FUNCTION_BLOCK PrintBools (* Basic Function Block Type *)
  (* Standard: 61499-2 *)
  (* Version 0.2, 2003-12-04, JHC, Rockwell Automation, Renamed for better indexing. *)
  (* Compiler header: package fb.rt.wago; *)
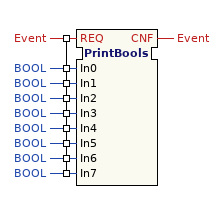
  EVENT_INPUT
    REQ WITH In0, In1, In2, In3, In4, In5, In6, In7; (* Normal Execution Request *)
  END_EVENT
  EVENT_OUTPUT
    CNF; (* Execution Confirmation *)
  END_EVENT
  VAR_INPUT
    In0 : BOOL := false; (* Input event qualifier *)
    In1 : BOOL := false; (* Input event qualifier *)
    In2 : BOOL := false; (* Input event qualifier *)
    In3 : BOOL := false; (* Input event qualifier *)
    In4 : BOOL := false; (* Input event qualifier *)
    In5 : BOOL := false; (* Input event qualifier *)
    In6 : BOOL := false; (* Input event qualifier *)
    In7 : BOOL := false; (* Input event qualifier *)
  END_VAR
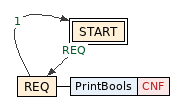
  EC_STATES
    START; (* Initial State *)
    REQ : PrintBools -> CNF; (* Normal execution *)
  END_STATES
  EC_TRANSITIONS
    START TO REQ := REQ;
    REQ TO START := 1;
  END_TRANSITIONS
  ALGORITHM PrintBools IN C: (* Normally executed algorithm *)
if( me->In0 ) printf("1"); else printf("0");
if( me->In1 ) printf("1"); else printf("0");
if( me->In2 ) printf("1"); else printf("0");
if( me->In3 ) printf("1"); else printf("0");
if( me->In4 ) printf("1"); else printf("0");
if( me->In5 ) printf("1"); else printf("0");
if( me->In6 ) printf("1"); else printf("0");
if( me->In7 ) printf("1"); else printf("0");
printf("\n");
  END_ALGORITHM
END_FUNCTION_BLOCK
